PROGRAM DebugMode
VAR
(* Common*)
	d_state: DINT;(*PowerOffState*)
	InitDone:BOOL;
	Busy: BOOL;
	fb_ton: TON;
	PowerState: INT;(*PowerOnState*)
	ton_t: TON;
(*Key Command*)
	LeftTopLinPositionNew:LREAL:=10;
	LeftTopLinVelocityNew:LREAL:=0.2;
	btn_LeftTopLinMove:BOOL;
	btn_LeftTopLinStop:BOOL;
	RightTopLinPositionNew:LREAL:=10;
	RightTopLinVelocityNew:LREAL:=0.2;
	btn_RightTopLinMove:BOOL;
	btn_RightTopLinStop:BOOL;
	LeftBottomLinPositionNew:LREAL:=10;
	LeftBottomLinVelocityNew:LREAL:=0.2;
	btn_LeftBottomLinMove:BOOL;
	btn_LeftBottomLinStop:BOOL;
	RightBottomLinPositionNew:LREAL:=10;
	RightBottomLinVelocityNew:LREAL:=0.2;
	btn_RightBottomLinMove:BOOL;
	btn_RightBottomLinStop:BOOL;
	
	
	LeftInLinPositionNew:LREAL:=10;
	LeftInLinVelocityNew:LREAL:=0.2;
	btn_LeftInLinMove:BOOL;
	btn_LeftInLinStop:BOOL;
	RightInLinPositionNew:LREAL:=10;
	RightInLinVelocityNew:LREAL:=0.2;
	btn_RightInLinMove:BOOL;
	btn_RightInLinStop:BOOL;
	LeftOutLinPositionNew:LREAL:=10;
	LeftOutLinVelocityNew:LREAL:=0.2;
	btn_LeftOutLinMove:BOOL;
	btn_LeftOutLinStop:BOOL;
	RightOutLinPositionNew:LREAL:=10;
	RightOutLinVelocityNew:LREAL:=0.2;
	btn_RightOutLinMove:BOOL;
	btn_RightOutLinStop:BOOL;
(*LeftTopLin*)
	fb_ton1_1:TON;
	fb_ton1_2:TON;
	LeftTopLinState:DINT;
	LeftTopLinBusy:BOOL;
	LeftTopLin_m_state: DINT;
	LeftTopLin_s_state: DINT;
(*RightTopLin*)
	fb_ton2_1:TON;
	fb_ton2_2:TON;
	RightTopLinState:DINT;
	RightTopLinBusy:BOOL;
	RightTopLin_m_state: DINT;
	RightTopLin_s_state: DINT;
(*LeftBottomLin*)
	fb_ton3_1:TON;
	fb_ton3_2:TON;
	LeftBottomLinState:DINT;
	LeftBottomLinBusy:BOOL;
	LeftBottomLin_m_state: DINT;
	LeftBottomLin_s_state: DINT;
(*RightBottomLin*)
	fb_ton4_1:TON;
	fb_ton4_2:TON;
	RightBottomLinState:DINT;
	RightBottomLinBusy:BOOL;
	RightBottomLin_m_state: DINT;
	RightBottomLin_s_state: DINT;
	
(*LeftInLin*)
	fb_ton5_1:TON;
	fb_ton5_2:TON;
	LeftInLinState:DINT;
	LeftInLinBusy:BOOL;
	LeftInLin_m_state: DINT;
	LeftInLin_s_state: DINT;
(*RightInLin*)
	fb_ton6_1:TON;
	fb_ton6_2:TON;
	RightInLinState:DINT;
	RightInLinBusy:BOOL;
	RightInLin_m_state: DINT;
	RightInLin_s_state: DINT;
(*LeftOutLin*)
	fb_ton7_1:TON;
	fb_ton7_2:TON;
	LeftOutLinState:DINT;
	LeftOutLinBusy:BOOL;
	LeftOutLin_m_state: DINT;
	LeftOutLin_s_state: DINT;
(*RightOutLin*)
	fb_ton8_1:TON;
	fb_ton8_2:TON;
	RightOutLinState:DINT;
	RightOutLinBusy:BOOL;
	RightOutLin_m_state: DINT;
	RightOutLin_s_state: DINT;


	btn_LeftTopStop: BOOL;
	(*¼ì²âµ½ÏÞÎ»£¬»Ö¸´Move×´Ì¬*)
	FTrig_ReachLS: F_TRIG;
	FTrig_btn_GapMove: F_TRIG;
END_VAR

(*********Monitor All Carrirt Position**********************)
A_MonitoringAllAxis();
(*********A_PosDiffDetection********************************)
A_PosDiffDetection();
(*********btn_PowerOn***************************************)
IF st_Power=1 THEN
	InitDone:=TRUE;
END_IF
IF btn_Power AND st_Power=0 THEN
	btn_PowerOn:=TRUE;
	btn_Power:=FALSE;
END_IF
IF btn_Power AND st_Power=1 THEN
	btn_PowerOff:=TRUE;
	btn_Power:=FALSE;
END_IF
(**********btn_PowerOn****************************************)
IF btn_PowerOn THEN
	A_PowerOn();
END_IF
IF btn_PowerOff THEN
	A_PowerOff();
END_IF

(**************btn_PowerOff*******************************)
IF btn_PowerOff THEN
	A_PowerOff();
END_IF

(**********************MOVE****************)
A_DebugMove();
(**********************STOP***************)
A_DebugStop();

FTrig_ReachLS(CLK:=Unreach_LS_Far AND Unreach_LS_Near);
IF FTrig_ReachLS.Q THEN
	btn_LeftTopLinStop:=TRUE;
	btn_RightTopLinStop:=TRUE;
	btn_LeftBottomLinStop:=TRUE;
	btn_RightBottomLinStop:=TRUE;
	btn_LeftInLinStop:=TRUE;
	btn_RightInLinStop:=TRUE;
	btn_LeftOutLinStop:=TRUE;
	btn_RightOutLinStop:=TRUE;
END_IF

ACTION A_DebugMove:
(*********************************************************************LeftTop_MOVE*****************************************************************)
IF InitDone THEN
	IF btn_LeftTopLinMove THEN
		CASE LeftTopLin_m_state OF
			0:
				FB_Move.Mode:=2;
				FB_Move.CoupleState:=st_Couple;	
				FB_Move.PowerState:=st_Power;	
				FB_Move.LeftTopMove:=TRUE;	
				FB_Move.LeftTopPosition:=LeftTopLinPositionNew;
				FB_Move.LeftTopVelocity:=LeftTopLinVelocityNew;	
				FB_Move();								
				LeftTopLin_m_state:=1;
			1:
				FB_Move();
				IF NOT FB_Move.LeftTopDone THEN
					LeftTopLin_m_state:=1;
					LED_Run:=TRUE;
				ELSE									
					LeftTopLin_m_state:=88;
				END_IF

			88:
				btn_LeftTopLinMove:=FALSE;
				LeftTopLin_m_state:=0;
				LED_Run:=FALSE;
		END_CASE
	END_IF
END_IF

(*********************************************************************RightTop_MOVE*****************************************************************)
IF InitDone THEN
	IF btn_RightTopLinMove THEN
		CASE RightTopLin_m_state OF
			0:
				FB_Move.Mode:=2;	
				FB_Move.CoupleState:=st_Couple;	
				FB_Move.PowerState:=st_Power;	
				FB_Move.RightTopMove:=TRUE;	
				FB_Move.RightTopPosition:=RightTopLinPositionNew;
				FB_Move.RightTopVelocity:=RightTopLinVelocityNew;
				FB_Move();
				RightTopLin_m_state:=1;
			1:
				FB_Move();
				IF NOT FB_Move.RightTopDone THEN
					RightTopLin_m_state:=1;
					LED_Run:=TRUE;
				ELSE
					RightTopLin_m_state:=88;
				END_IF

			88:
				btn_RightTopLinMove:=FALSE;	
				RightTopLin_m_state:=0;
				LED_Run:=FALSE;
		END_CASE
	END_IF
END_IF

(*********************************************************************LeftBottom_MOVE*****************************************************************)
IF InitDone THEN
	IF btn_LeftBottomLinMove THEN
		CASE LeftBottomLin_m_state OF
			0:
				FB_Move.Mode:=2;	
				FB_Move.CoupleState:=st_Couple;	
				FB_Move.PowerState:=st_Power;
				FB_Move.LeftBottomMove:=TRUE;
				FB_Move.LeftBottomPosition:=LeftBottomLinPositionNew;
				FB_Move.LeftBottomVelocity:=LeftBottomLinVelocityNew;
				FB_Move();	
				LeftBottomLin_m_state:=1;
			1:
				FB_Move();
				IF NOT FB_Move.LeftBottomDone THEN	
					LeftBottomLin_m_state:=1;
					LED_Run:=TRUE;
				ELSE
					LeftBottomLin_m_state:=88;
				END_IF

			88:
				btn_LeftBottomLinMove:=FALSE;
				LeftBottomLin_m_state:=0;
				LED_Run:=FALSE;
		END_CASE
	END_IF
END_IF

(*********************************************************************RightBottom_MOVE*****************************************************************)
IF InitDone THEN
	IF btn_RightBottomLinMove THEN
		CASE RightBottomLin_m_state OF
			0:
				FB_Move.Mode:=2;
				FB_Move.CoupleState:=st_Couple;	
				FB_Move.PowerState:=st_Power;
				FB_Move.RightBottomMove:=TRUE;
				FB_Move.RightBottomPosition:=RightBottomLinPositionNew;
				FB_Move.RightBottomVelocity:=RightBottomLinVelocityNew;	
				FB_Move();	
				RightBottomLin_m_state:=1;
			1:
				FB_Move();
				IF NOT FB_Move.RightBottomDone THEN	
					RightBottomLin_m_state:=1;
					LED_Run:=TRUE;
				ELSE	
					RightBottomLin_m_state:=88;
				END_IF

			88:
				btn_RightBottomLinMove:=FALSE;
				RightBottomLin_m_state:=0;
				LED_Run:=FALSE;
		END_CASE
	END_IF
END_IF

(*********************************************************************LeftIn_MOVE*****************************************************************)
IF InitDone THEN
	IF btn_LeftInLinMove THEN
		CASE LeftInLin_m_state OF
			0:
				FB_Move.Mode:=2;
				FB_Move.CoupleState:=st_Couple;	
				FB_Move.PowerState:=st_Power;	
				FB_Move.LeftInMove:=TRUE;	
				FB_Move.LeftInPosition:=LeftInLinPositionNew;
				FB_Move.LeftInVelocity:=LeftInLinVelocityNew;	
				FB_Move();								
				LeftInLin_m_state:=1;
			1:
				FB_Move();
				IF NOT FB_Move.LeftInDone THEN
					LeftInLin_m_state:=1;
					LED_Run:=TRUE;
				ELSE									
					LeftInLin_m_state:=88;
				END_IF

			88:
				btn_LeftInLinMove:=FALSE;
				LeftInLin_m_state:=0;
				LED_Run:=FALSE;
		END_CASE
	END_IF
END_IF

(*********************************************************************RightIn_MOVE*****************************************************************)
IF InitDone THEN
	IF btn_RightInLinMove THEN
		CASE RightInLin_m_state OF
			0:
				FB_Move.Mode:=2;	
				FB_Move.CoupleState:=st_Couple;	
				FB_Move.PowerState:=st_Power;	
				FB_Move.RightInMove:=TRUE;	
				FB_Move.RightInPosition:=RightInLinPositionNew;
				FB_Move.RightInVelocity:=RightInLinVelocityNew;
				FB_Move();
				RightInLin_m_state:=1;
			1:
				FB_Move();
				IF NOT FB_Move.RightInDone THEN
					RightInLin_m_state:=1;
					LED_Run:=TRUE;
				ELSE
					RightInLin_m_state:=88;
				END_IF

			88:
				btn_RightInLinMove:=FALSE;	
				RightInLin_m_state:=0;
				LED_Run:=FALSE;
		END_CASE
	END_IF
END_IF

(*********************************************************************LeftOut_MOVE*****************************************************************)
IF InitDone THEN
	IF btn_LeftOutLinMove THEN
		CASE LeftOutLin_m_state OF
			0:
				FB_Move.Mode:=2;	
				FB_Move.CoupleState:=st_Couple;	
				FB_Move.PowerState:=st_Power;
				FB_Move.LeftOutMove:=TRUE;
				FB_Move.LeftOutPosition:=LeftOutLinPositionNew;
				FB_Move.LeftOutVelocity:=LeftOutLinVelocityNew;
				FB_Move();	
				LeftOutLin_m_state:=1;
			1:
				FB_Move();
				IF NOT FB_Move.LeftOutDone THEN	
					LeftOutLin_m_state:=1;
					LED_Run:=TRUE;
				ELSE
					LeftOutLin_m_state:=88;
				END_IF

			88:
				btn_LeftOutLinMove:=FALSE;
				LeftOutLin_m_state:=0;
				LED_Run:=FALSE;
		END_CASE
	END_IF
END_IF

(*********************************************************************RightOut_MOVE*****************************************************************)
IF InitDone THEN
	IF btn_RightOutLinMove THEN
		CASE RightOutLin_m_state OF
			0:
				FB_Move.Mode:=2;
				FB_Move.CoupleState:=st_Couple;	
				FB_Move.PowerState:=st_Power;
				FB_Move.RightOutMove:=TRUE;
				FB_Move.RightOutPosition:=RightOutLinPositionNew;
				FB_Move.RightOutVelocity:=RightOutLinVelocityNew;	
				FB_Move();	
				RightOutLin_m_state:=1;
			1:
				FB_Move();
				IF NOT FB_Move.RightOutDone THEN	
					RightOutLin_m_state:=1;
					LED_Run:=TRUE;
				ELSE	
					RightOutLin_m_state:=88;
				END_IF

			88:
				btn_RightOutLinMove:=FALSE;
				RightOutLin_m_state:=0;
				LED_Run:=FALSE;
		END_CASE
	END_IF
END_IF
END_ACTION

ACTION A_DebugStop:
(*******************************************************************LeftTop_STOP********************************************************************)
IF btn_LeftTopLinStop THEN
	LED_Run:=FALSE;
	FB_Move.LeftTopReset:=TRUE;	
	FB_Move();	
	btn_LeftTopLinMove:=FALSE;	
	LeftTopLin_m_state:=0;	
	CASE LeftTopLin_s_state OF
			0:
				FB_Stop.Mode:=2;
				FB_Stop.CoupleState:=st_Couple;	
				FB_Stop.PowerState:=st_Power;	
				FB_Stop.LeftTopStop:=TRUE;
				FB_Stop();	
				LeftTopLin_s_state:=1;
			1:
				FB_Stop();
				IF NOT FB_Stop.LeftTopDone THEN	
					LeftTopLin_s_state:=1;
				ELSE
					LeftTopLin_s_state:=88;
				END_IF
			88:
				btn_LeftTopLinStop:=FALSE;	
				FB_Move.LeftTopReset:=FALSE;	
				LeftTopLin_s_state:=0;
		END_CASE

END_IF

(*******************************************************************RightTop_STOP********************************************************************)
IF btn_RightTopLinStop THEN
	LED_Run:=FALSE;
	FB_Move.RightTopReset:=TRUE;
	FB_Move();
	btn_RightTopLinMove:=FALSE;	
	RightTopLin_m_state:=0;		
	CASE RightTopLin_s_state OF
			0:
				FB_Stop.Mode:=2;
				FB_Stop.CoupleState:=st_Couple;
				FB_Stop.PowerState:=st_Power;
				FB_Stop.RightTopStop:=TRUE;
				FB_Stop();
				RightTopLin_s_state:=1;
			1:
				FB_Stop();
				IF NOT FB_Stop.RightTopDone THEN
					RightTopLin_s_state:=1;
				ELSE	
					RightTopLin_s_state:=88;
				END_IF
			88:
				btn_RightTopLinStop:=FALSE;	
				FB_Move.RightTopReset:=FALSE;
				RightTopLin_s_state:=0;
		END_CASE

END_IF

(*******************************************************************LeftBottom_STOP********************************************************************)
IF btn_LeftBottomLinStop THEN
	LED_Run:=FALSE;
	FB_Move.LeftBottomReset:=TRUE;
	FB_Move();						
	btn_LeftBottomLinMove:=FALSE;		
	LeftBottomLin_m_state:=0;		
	CASE LeftBottomLin_s_state OF
			0:
				FB_Stop.Mode:=2;
				FB_Stop.CoupleState:=st_Couple;
				FB_Stop.PowerState:=st_Power;
				FB_Stop.LeftBottomStop:=TRUE;	
				FB_Stop();	
				LeftBottomLin_s_state:=1;
			1:
				FB_Stop();
				IF NOT FB_Stop.LeftBottomDone THEN
					LeftBottomLin_s_state:=1;
				ELSE
					LeftBottomLin_s_state:=88;
				END_IF
			88:
				btn_LeftBottomLinStop:=FALSE;
				FB_Move.LeftBottomReset:=FALSE;	
				LeftBottomLin_s_state:=0;
		END_CASE

END_IF

(*******************************************************************RightBottom_STOP********************************************************************)
IF btn_RightBottomLinStop THEN
	LED_Run:=FALSE;
	FB_Move.RightBottomReset:=TRUE;
	FB_Move();	
	btn_RightBottomLinMove:=FALSE;
	RightBottomLin_m_state:=0;	
	CASE RightBottomLin_s_state OF
			0:
				FB_Stop.Mode:=2;
				FB_Stop.CoupleState:=st_Couple;	
				FB_Stop.PowerState:=st_Power;
				FB_Stop.RightBottomStop:=TRUE;	
				FB_Stop();
				RightBottomLin_s_state:=1;
			1:
				FB_Stop();
				IF NOT FB_Stop.RightBottomDone THEN
					RightBottomLin_s_state:=1;
				ELSE
					RightBottomLin_s_state:=88;
				END_IF
			88:
				btn_RightBottomLinStop:=FALSE;
				FB_Move.RightBottomReset:=FALSE;
				RightBottomLin_s_state:=0;
		END_CASE

END_IF

(*******************************************************************LeftIn_STOP********************************************************************)
IF btn_LeftInLinStop THEN
	LED_Run:=FALSE;
	FB_Move.LeftInReset:=TRUE;	
	FB_Move();	
	btn_LeftInLinMove:=FALSE;	
	LeftInLin_m_state:=0;	
	CASE LeftInLin_s_state OF
			0:
				FB_Stop.Mode:=2;
				FB_Stop.CoupleState:=st_Couple;	
				FB_Stop.PowerState:=st_Power;	
				FB_Stop.LeftInStop:=TRUE;
				FB_Stop();	
				LeftInLin_s_state:=1;
			1:
				FB_Stop();
				IF NOT FB_Stop.LeftInDone THEN	
					LeftInLin_s_state:=1;
				ELSE
					LeftInLin_s_state:=88;
				END_IF
			88:
				btn_LeftInLinStop:=FALSE;	
				FB_Move.LeftInReset:=FALSE;	
				LeftInLin_s_state:=0;
		END_CASE

END_IF

(*******************************************************************RightIn_STOP********************************************************************)
IF btn_RightInLinStop THEN
	LED_Run:=FALSE;
	FB_Move.RightInReset:=TRUE;
	FB_Move();
	btn_RightInLinMove:=FALSE;	
	RightInLin_m_state:=0;		
	CASE RightInLin_s_state OF
			0:
				FB_Stop.Mode:=2;
				FB_Stop.CoupleState:=st_Couple;
				FB_Stop.PowerState:=st_Power;
				FB_Stop.RightInStop:=TRUE;
				FB_Stop();
				RightInLin_s_state:=1;
			1:
				FB_Stop();
				IF NOT FB_Stop.RightInDone THEN
					RightInLin_s_state:=1;
				ELSE	
					RightInLin_s_state:=88;
				END_IF
			88:
				btn_RightInLinStop:=FALSE;	
				FB_Move.RightInReset:=FALSE;
				RightInLin_s_state:=0;
		END_CASE

END_IF

(*******************************************************************LeftOut_STOP********************************************************************)
IF btn_LeftOutLinStop THEN
	LED_Run:=FALSE;
	FB_Move.LeftOutReset:=TRUE;
	FB_Move();						
	btn_LeftOutLinMove:=FALSE;		
	LeftOutLin_m_state:=0;		
	CASE LeftOutLin_s_state OF
			0:
				FB_Stop.Mode:=2;
				FB_Stop.CoupleState:=st_Couple;
				FB_Stop.PowerState:=st_Power;
				FB_Stop.LeftOutStop:=TRUE;	
				FB_Stop();	
				LeftOutLin_s_state:=1;
			1:
				FB_Stop();
				IF NOT FB_Stop.LeftOutDone THEN
					LeftOutLin_s_state:=1;
				ELSE
					LeftOutLin_s_state:=88;
				END_IF
			88:
				btn_LeftOutLinStop:=FALSE;
				FB_Move.LeftOutReset:=FALSE;	
				LeftOutLin_s_state:=0;
		END_CASE

END_IF

(*******************************************************************RightOut_STOP********************************************************************)
IF btn_RightOutLinStop THEN
	LED_Run:=FALSE;
	FB_Move.RightOutReset:=TRUE;
	FB_Move();	
	btn_RightOutLinMove:=FALSE;
	RightOutLin_m_state:=0;	
	CASE RightOutLin_s_state OF
			0:
				FB_Stop.Mode:=2;
				FB_Stop.CoupleState:=st_Couple;	
				FB_Stop.PowerState:=st_Power;
				FB_Stop.RightOutStop:=TRUE;	
				FB_Stop();
				RightOutLin_s_state:=1;
			1:
				FB_Stop();
				IF NOT FB_Stop.RightOutDone THEN
					RightOutLin_s_state:=1;
				ELSE
					RightOutLin_s_state:=88;
				END_IF
			88:
				btn_RightOutLinStop:=FALSE;
				FB_Move.RightOutReset:=FALSE;
				RightOutLin_s_state:=0;
		END_CASE

END_IF
END_ACTION

ACTION A_monitoringAllAxis:
(*************************************************************************************2.4Öá¹âÕ¤³ßÎ»ÖÃ¡¢ËÙ¶È¶Ô±È¼ì²é**********************************************************************)
IF st_power<>0 THEN

IF ABS(Pos_LeftTopLin-Pos_LeftBottomLin)>Threshold_TBLeftPos_Debug  THEN
		btn_LeftTopLinStop:=TRUE;
		btn_RightTopLinStop:=TRUE;
		btn_LeftBottomLinStop:=TRUE;
		btn_RightBottomLInStop:=TRUE;
		FB_PlcEmergencyStop();
		Error:=TRUE;
		ErrorID:=11;
		LED_Error:=TRUE;
END_IF

IF ABS(Pos_RightTopLin-Pos_RightBottomLin)>Threshold_TBRightPos_Debug  THEN
		btn_LeftTopLinStop:=TRUE;
		btn_RightTopLinStop:=TRUE;
		btn_LeftBottomLinStop:=TRUE;
		btn_RightBottomLInStop:=TRUE;
		FB_PlcEmergencyStop();
		Error:=TRUE;
		ErrorID:=12;
		LED_Error:=TRUE;
END_IF

IF ABS(Pos_LeftTopLin-Pos_RightTopLin)>Threshold_TopPos_Debug  THEN
		btn_LeftTopLinStop:=TRUE;
		btn_RightTopLinStop:=TRUE;
		btn_LeftBottomLinStop:=TRUE;
		btn_RightBottomLInStop:=TRUE;
		FB_PlcEmergencyStop();
		Error:=TRUE;
		ErrorID:=13;
		LED_Error:=TRUE;
END_IF

IF ABS(Pos_LeftBottomLin-Pos_RightBottomLin)>Threshold_BottomPos_Debug  THEN
		btn_LeftTopLinStop:=TRUE;
		btn_RightTopLinStop:=TRUE;
		btn_LeftBottomLinStop:=TRUE;
		btn_RightBottomLInStop:=TRUE;
		FB_PlcEmergencyStop();
		Error:=TRUE;
		ErrorID:=14;
		LED_Error:=TRUE;
END_IF
//

IF ABS(Pos_LeftInLin-Pos_LeftOutLin)>Threshold_IOLeftPos_Debug  THEN
		btn_LeftInLinStop:=TRUE;
		btn_RightInLinStop:=TRUE;
		btn_LeftOutLinStop:=TRUE;
		btn_RightOutLInStop:=TRUE;
		FB_PlcEmergencyStop();
		Error:=TRUE;
		ErrorID:=15;
		LED_Error:=TRUE;
END_IF

IF ABS(Pos_RightInLin-Pos_RightOutLin)>Threshold_IORightPos_Debug  THEN
		btn_LeftInLinStop:=TRUE;
		btn_RightInLinStop:=TRUE;
		btn_LeftOutLinStop:=TRUE;
		btn_RightOutLInStop:=TRUE;
		FB_PlcEmergencyStop();
		Error:=TRUE;
		ErrorID:=16;
		LED_Error:=TRUE;
END_IF

IF ABS(Pos_LeftInLin-Pos_RightInLin)>Threshold_InPos_Debug  THEN
		btn_LeftInLinStop:=TRUE;
		btn_RightInLinStop:=TRUE;
		btn_LeftOutLinStop:=TRUE;
		btn_RightOutLInStop:=TRUE;
		FB_PlcEmergencyStop();
		Error:=TRUE;
		ErrorID:=17;
		LED_Error:=TRUE;
END_IF

IF ABS(Pos_LeftOutLin-Pos_RightOutLin)>Threshold_OutPos_Debug  THEN
		btn_LeftInLinStop:=TRUE;
		btn_RightInLinStop:=TRUE;
		btn_LeftOutLinStop:=TRUE;
		btn_RightOutLInStop:=TRUE;
		FB_PlcEmergencyStop();
		Error:=TRUE;
		ErrorID:=18;
		LED_Error:=TRUE;
END_IF
END_IF
END_ACTION

ACTION A_PosDiffDetection:
IF ABS(PosDiff_LeftTopLin_actual-PosDiff_RightTopLin_actual)>0.2 THEN
	ErrorID:=51;
	Error:=TRUE;
	btn_LeftTopLinStop:=TRUE;
	btn_RightTopLinStop:=TRUE;
	btn_LeftBottomLinStop:=TRUE;
	btn_RightBottomLInStop:=TRUE;
	FB_PlcEmergencyStop();
	LED_Error:=TRUE;
ELSIF ABS(PosDiff_LeftBottomLin_actual-PosDiff_RightBottomLin_actual)>0.2 THEN
	ErrorID:=52;
	Error:=TRUE;
	btn_LeftTopLinStop:=TRUE;
	btn_RightTopLinStop:=TRUE;
	btn_LeftBottomLinStop:=TRUE;
	btn_RightBottomLInStop:=TRUE;
	FB_PlcEmergencyStop();
	LED_Error:=TRUE;
END_IF

IF ABS(PosDiff_LeftInLin_actual-PosDiff_RightInLin_actual)>0.2 THEN
	ErrorID:=53;
	Error:=TRUE;
	btn_LeftInLinStop:=TRUE;
	btn_RightInLinStop:=TRUE;
	btn_LeftOutLinStop:=TRUE;
	btn_RightOutLInStop:=TRUE;
	FB_PlcEmergencyStop();
	LED_Error:=TRUE;
ELSIF ABS(PosDiff_LeftOutLin_actual-PosDiff_RightOutLin_actual)>0.2 THEN
	ErrorID:=54;
	Error:=TRUE;
	btn_LeftInLinStop:=TRUE;
	btn_RightInLinStop:=TRUE;
	btn_LeftOutLinStop:=TRUE;
	btn_RightOutLInStop:=TRUE;
	FB_PlcEmergencyStop();
	LED_Error:=TRUE;
END_IF
END_ACTION

ACTION A_PowerOff:
CASE d_state OF
		0:(*PowerOff*)
			FB_Power(Off:=TRUE);
				d_state:=1;
		1:
			IF NOT FB_power.OffStatus THEN
				d_state:=1;
			ELSE
				d_state:=88;
			END_IF
		88:(*ResetAllState*)
			btn_PowerOn:=FALSE;
			btn_PowerOff:=FALSE;
			ton_t.IN:=FALSE;
			InitDone:=FALSE;
			Error:=FALSE;
			ErrorID:=0;
			d_state:=0;

			btn_LeftTopLinMove:=FALSE;
			btn_LeftTopLinStop:=FALSE;
			fb_ton1_1.IN:=FALSE;
			fb_ton1_2.IN:=FALSE;
			LeftTopLinState:=0;
			LeftTopLinBusy:=FALSE;
			LeftTopLin_m_state:=0;
			LeftTopLin_s_state:=0;

			btn_RightTopLinMove:=FALSE;
			btn_RightTopLinStop:=FALSE;
			fb_ton2_1.IN:=FALSE;
			fb_ton2_2.IN:=FALSE;
			RightTopLinState:=0;
			RightTopLinBusy:=FALSE;
			RightTopLin_m_state:=0;
			RightTopLin_s_state:=0;

			btn_LeftBottomLinMove:=FALSE;
			btn_LeftBottomLinStop:=FALSE;
			fb_ton3_1.IN:=FALSE;
			fb_ton3_2.IN:=FALSE;
			LeftBottomLinState:=0;
			LeftBottomLinBusy:=FALSE;
			LeftBottomLin_m_state:=0;
			LeftBottomLin_s_state:=0;

			btn_RightBottomLinMove:=FALSE;
			btn_RightBottomLinStop:=FALSE;
			fb_ton4_1.IN:=FALSE;
			fb_ton4_2.IN:=FALSE;
			RightBottomLinState:=0;
			RightBottomLinBusy:=FALSE;
			RightBottomLin_m_state:=0;
			RightBottomLin_s_state:=0;
			
			btn_LeftInLinMove:=FALSE;
			btn_LeftInLinStop:=FALSE;
			fb_ton5_1.IN:=FALSE;
			fb_ton5_2.IN:=FALSE;
			LeftInLinState:=0;
			LeftInLinBusy:=FALSE;
			LeftInLin_m_state:=0;
			LeftInLin_s_state:=0;

			btn_RightInLinMove:=FALSE;
			btn_RightInLinStop:=FALSE;
			fb_ton6_1.IN:=FALSE;
			fb_ton6_2.IN:=FALSE;
			RightInLinState:=0;
			RightInLinBusy:=FALSE;
			RightInLin_m_state:=0;
			RightInLin_s_state:=0;

			btn_LeftOutLinMove:=FALSE;
			btn_LeftOutLinStop:=FALSE;
			fb_ton7_1.IN:=FALSE;
			fb_ton7_2.IN:=FALSE;
			LeftBottomLinState:=0;
			LeftOutLinBusy:=FALSE;
			LeftOutLin_m_state:=0;
			LeftOutLin_s_state:=0;

			btn_RightOutLinMove:=FALSE;
			btn_RightOutLinStop:=FALSE;
			fb_ton8_1.IN:=FALSE;
			fb_ton8_2.IN:=FALSE;
			RightOutLinState:=0;
			RightOutLinBusy:=FALSE;
			RightOutLin_m_state:=0;
			RightOutLin_s_state:=0;

		LED_Error:=FALSE;
		LED_Run:=FALSE;

END_CASE
END_ACTION

ACTION A_PowerOn:
fb_ton(PT:=T#0.5S);
CASE PowerState OF
	0:	(*FB_Power_On*)
		FB_Power(On:=TRUE);
		fb_ton.IN:=TRUE;
		PowerState:=1;
	1:	(*wait*)
		FB_power();
		IF NOT FB_power.OnStatus THEN		(*FB_Power_OnÃ»ÓÐÖ´ÐÐÍê£¬wait£¬³¬Ê±FB Error*)
			IF NOT fb_ton.Q THEN
				PowerState:=1;
			ELSE
				ErrorID:=1;
				PowerState:=99;
			END_IF
		ELSE
			PowerState:=88;
		END_IF
	88:	(*All Done*)
		btn_PowerOn:=FALSE;
		PowerState:=0;
		Error:=FALSE;
		ErrorID:=0;
		Busy:=FALSE;
		InitDone:=TRUE;
		FB_power.On:=FALSE;
		fb_ton.IN:=FALSE;
		LED_Error:=FALSE;
	99:
		btn_PowerOn:=FALSE;
		PowerState:=99;
		Error:=TRUE;
		Busy:=FALSE;
		InitDone:=FALSE;
		FB_Power.On:=FALSE;
		fb_ton.IN:=FALSE;
		LED_Error:=TRUE;
END_CASE
END_ACTION

END_PROGRAM

(* stored: Version 1.1.0.1, ProductVersion 3.1.4024.6
   POU DebugMode: Id {9c1b652b-c28b-4723-806b-1a1456d9a5fb}, SpecialFunc None
   Action A_DebugMove: Id {688a6355-0b41-43f8-8d7d-2cc411073576}
   Action A_DebugStop: Id {00c13c2f-a1d0-477f-a2a0-6eec97b28739}
   Action A_monitoringAllAxis: Id {d1a34df5-69b1-4771-bf4a-eb30f477489b}
   Action A_PosDiffDetection: Id {0b914de3-5a16-4135-8c47-916309d8d3da}
   Action A_PowerOff: Id {e677fe86-edfe-48c4-ba29-b932f9bd11d2}
   Action A_PowerOn: Id {3be612a8-046c-45b5-ad28-b2fb90dcb4f1} *)
